// TwinCAT 3 PLC project Untitled1
// ProgramVersion: 3.1.4024.0
// libraries:
//   Tc2_Standard, * (Beckhoff Automation GmbH)
//   Tc2_System, * (Beckhoff Automation GmbH)
//   Tc3_Module, * (Beckhoff Automation GmbH)
//   TcUnit, * (www.tcunit.org)
// project tree:
//   FileHandle/ FB_FileHandle.TcPOU
//   / PlcTask.TcTTO
//   POUs/ MAIN.TcPOU
//   Test/ FileHandle_Test.TcPOU, POU_Test.TcPOU
// real-time tasks:
//   TASK PlcTask: cycle T#10ms, priority 20, ADS port 350

CONFIGURATION Untitled1
    RESOURCE PLC ON TwinCAT3
        TASK PlcTask(INTERVAL := T#10ms, PRIORITY := 20);
        PROGRAM MAIN WITH PlcTask : MAIN;
    END_RESOURCE
END_CONFIGURATION

// ---- POUs/MAIN.TcPOU
PROGRAM MAIN
VAR
	
END_VAR

POU_Test();

END_PROGRAM

// ---- Test/POU_Test.TcPOU
PROGRAM POU_Test
VAR
	fbFileHandle_Test: FileHandle_Test;
END_VAR

TcUnit.RUN();

END_PROGRAM

// ---- Test/FileHandle_Test.TcPOU
FUNCTION_BLOCK FileHandle_Test EXTENDS TcUnit.FB_TestSuite
VAR
	{attribute 'old_input_assignments' := ''}
	fbFilehandle: FB_FileHandle('C:\logtest', 'test.txt');
END_VAR

fileopen();
filewriteHelloWorld();
fileclose();

METHOD fileclose
VAR_INST
	Timer : TON := (PT := T#10S);
	Actual : BOOL;
	step : INT;
	ExpectedValue : BOOL := TRUE;
END_VAR
IF TEST_ORDERED('fileclose') THEN
	Timer(IN:=TRUE);
	fbFilehandle.M_FileClose();
	
	Actual := fbFilehandle.isFileClosed;
	
	IF Timer.Q OR Actual = ExpectedValue THEN
		AssertEquals(Expected := ExpectedValue, Actual := Actual, Message:= 'File is not closed');
		TEST_FINISHED();
	END_IF
END_IF
END_METHOD

METHOD fileopen
VAR_INST
	Timer : TON := (PT := T#10S);
	ExpectedValue : BOOL := TRUE;
	Actual : BOOL;

END_VAR
IF TEST_ORDERED('fileopen') THEN
	Timer(IN:=TRUE);
	fbFilehandle.M_FileOpen();
	Actual := fbFilehandle.isFileOpened;
	
	IF Timer.Q OR fbFilehandle.isFileOpened THEN
		AssertEquals(Expected := ExpectedValue, Actual := Actual, Message:= 'File is not opened');
		TEST_FINISHED();
	END_IF
END_IF
END_METHOD

METHOD filewriteHelloWorld
VAR_INST
	Timer : TON := (PT := T#10S);
	ExpectedValue : STRING := '';
	Actual : STRING;
	step : INT;
END_VAR
IF TEST_ORDERED('filewriteHelloWorld') THEN
	Timer(IN:=TRUE);
	CASE step OF
		0:
			fbFilehandle.P_SomethingToWrite := 'Hello world';
			step := 10;
		10:
			fbFilehandle.M_FileWrite();		
	END_CASE
	
	Actual := fbFilehandle.P_SomethingToWrite;
	
	IF Timer.Q OR Actual ='' THEN
		AssertEquals(Expected := ExpectedValue, Actual := Actual, Message:= 'File is not written');
		TEST_FINISHED();
	END_IF
END_IF
END_METHOD

END_FUNCTION_BLOCK

// ---- FileHandle/FB_FileHandle.TcPOU
FUNCTION_BLOCK FB_FileHandle
VAR
	_sNetID: T_AmsNetId;
	_ErrorMessage: STRING;
	_bError: BOOL;
	_bFileOpened: BOOL;
	_bFileClosed: BOOL;
	_sWrite: STRING;
	_bDirectoryCreated: BOOL;
	sFileName: STRING;
	sDirectory: STRING;
	hFile: UINT;
	fbCreateDirectory: FB_CreateDir;
	fbFileOpen: FB_FileOpen;
	fbFileWrite: FB_FileWrite;
	fbFileClose: FB_FileClose;
END_VAR

METHOD FB_init : BOOL
VAR_INPUT
	/// if TRUE, the retain variables are initialized (warm start / cold start)
	bInitRetains: BOOL;
	/// if TRUE, the instance afterwards gets moved into the copy code (online change)
	bInCopyCode: BOOL;
	Directory: STRING;
	FileName: STRING;
END_VAR
M_SetPath(Directory, FileName);
END_METHOD

PROPERTY isErrorOccured : BOOL
GET
isErrorOccured := This^._bError;
END_GET
END_PROPERTY

PROPERTY isFileClosed : BOOL
GET
isFileClosed := This^._bFileClosed;
END_GET
END_PROPERTY

PROPERTY isFileOpened : BOOL
GET
isFileOpened := This^._bFileOpened;
END_GET
END_PROPERTY

METHOD M_FileClose
fbFileClose(
	sNetId:= _sNetId, 
	hFile:= hFile, 
	bExecute:= TRUE, 
	tTimeout:= , 
	bBusy=> , 
	bError=> , 
	nErrId=> );
	
IF fbFileClose.bError THEN
	_ErrorMessage := CONCAT('FileOpen Failed ErrID = ', UDINT_TO_STRING(fbFileClose.nErrId));
	_bError := TRUE;
	fbFileClose(bExecute := FALSE);
	Return;
END_IF

IF fbFileClose.bBusy THEN
	RETURN;
ELSE
	_bFileClosed := TRUE;
	_bFileOpened := FALSE;
END_IF
END_METHOD

METHOD M_FileOpen
IF NOT _bDirectoryCreated THEN
	fbCreateDirectory(sPathName := THIS^.sDirectory ,bExecute := TRUE);
	
	IF fbCreateDirectory.bBusy THEN
		_bDirectoryCreated := FALSE;
		RETURN;	
	ELSE 
		fbCreateDirectory(bExecute := FALSE);
		_bDirectoryCreated := TRUE;
	END_IF
ELSE
	fbFileOpen(
		sNetId:= , 
		sPathName:= P_FilePath, 
		nMode:= FOPEN_MODEAPPEND OR FOPEN_MODETEXT , 
		ePath:=PATH_GENERIC, 
		bExecute:= TRUE, 
		tTimeout:= , 
		bBusy=> , 
		bError=> , 
		nErrId=> , 
		hFile=> hFile);
	
	IF fbFileOpen.bError THEN
		_ErrorMessage := CONCAT('FileOpen Failed ErrID = ', UDINT_TO_STRING(fbFileOpen.nErrId));
		RETURN;
	END_IF
		
	IF fbFileOpen.bBusy THEN
		RETURN;
	ELSE
		fbFileOpen(bExecute := FALSE);
		_bFileOpened := TRUE;
		_bFileClosed := FALSE;
	END_IF
END_IF
END_METHOD

METHOD M_FileWrite
IF _sWrite <> '' THEN
	fbFileWrite(
		sNetId:= _sNetID, 
		hFile:= hFile, 
		pWriteBuff:= ADR(_sWrite) , 
		cbWriteLen:= INT_TO_UDINT(LEN(_sWrite)), 
		bExecute:= TRUE, 
		tTimeout:= , 
		bBusy=> , 
		bError=> , 
		nErrId=> , 
		cbWrite=> );
		
	IF fbFileWrite.bError THEN
		_ErrorMessage := CONCAT('FileWrite Failed ErrID = ', UDINT_TO_STRING(fbFileWrite.nErrId));
		Return;
	END_IF
	
	IF fbFileWrite.bBusy THEN
		RETURN;
	ELSE
		fbFileWrite(bExecute := FALSE);
		_sWrite := '';  //Reset sWrite after file write
	END_IF
END_IF
END_METHOD

METHOD PRIVATE M_SetPath
VAR_INPUT
	sDirectory: STRING;
	sFileName: STRING;
END_VAR
THIS^.sDirectory := sDirectory;
THIS^.sFileName := sFileName;
END_METHOD

PROPERTY P_ErrorMessage : T_Maxstring
GET
P_ErrorMessage := _ErrorMessage;
END_GET
END_PROPERTY

PROPERTY P_FilePath : STRING
GET
P_FilePath := CONCAT(This^.sDirectory, CONCAT('/', This^.sFileName));
END_GET
END_PROPERTY

PROPERTY P_sNetID : T_AmsNetID
GET
P_sNetID := This^._sNetID;
END_GET
SET
 This^._sNetID :=P_sNetID;
END_SET
END_PROPERTY

PROPERTY P_SomethingToWrite : T_Maxstring
GET
P_SomethingToWrite:= This^._sWrite ;
END_GET
SET
This^._sWrite := P_SomethingToWrite;
END_SET
END_PROPERTY

END_FUNCTION_BLOCK
